// TIA Portal project "Scena_pick_place" (V16)
// Vorlageprojekt für das Buch mit Zielsystem S7-1200

(* hardware
DEVICE "S7-1200-Station_1"  S7-1200 Station
   slot 0: "Baugruppenträger_0"  Rack  V1.0
   slot 1: "PLC_1"  CPU 1211C DC/DC/DC  6ES7 211-1AE40-0XB0  V4.1
*)

// ===== PLC "PLC_1"  CPU 1211C DC/DC/DC =====

VAR_GLOBAL   // PLC tag table "Standard-Variablentabelle"
   "Entry_Conveyor" AT %A0.0 : Bool;
   "Auto" AT %E0.0 : Bool;
   "Emergency_stop" AT %E0.1 : Bool;
   "Item_at_entry" AT %I0.2 : Bool;
   "Item_at_exit" AT %I0.3 : Bool;
   "Item_detected" AT %I0.4 : Bool;
   "Manual" AT %I0.5 : Bool;
   "Moving_x" AT %I0.6 : Bool;
   "Moving_z" AT %I0.7 : Bool;
   "Exit_conveyor" AT %Q0.1 : Bool;
   "Grab" AT %Q0.2 : Bool;
   "Move_x" AT %Q0.3 : Bool;
   "Move_z" AT %Q0.4 : Bool;
   "Reset" AT %I1.0 : Bool;
   "Start" AT %I1.1 : Bool;
   "Stop" AT %I1.2 : Bool;
   "Reset_light" AT %Q0.5 : Bool;
   "Start_light" AT %Q0.6 : Bool;
   "Stop_light" AT %Q0.7 : Bool;
   "Tag_1" AT %M0.0 : Bool;
   "Tag_2" AT %M0.1 : Bool;
   "Tag_3" AT %M0.2 : Bool;
   "Tag_4" AT %M0.3 : Bool;
   "Tag_5" AT %M0.4 : Bool;
   "Tag_6" AT %M0.5 : Bool;
   "Counter" AT %QD30 : DInt;
END_VAR

FUNCTION "MHJ-PLC-Lab-Function-S71200" : Void   // FC9000, SCL
{ S7_Optimized_Access := 'TRUE' }
VERSION : 0.1
   VAR_TEMP
      rdTimeReturn : Int;
      outputTime : DTL;
      SyncVal : Byte;
      forVal : Int;
      forVal_2 : Int;
      Value : Byte;
   END_VAR
   VAR CONSTANT
      CompVal : Byte := 16#34;
      Value_01 : Byte := 16#11;
      Value_01_DW : DWord := 16#A165_D992;
      Value_02_DW : DWord := 16#58BE_4401;
   END_VAR
BEGIN

   #Value:=PEEK(area := 16#82,
        dbNumber := 0,
        byteOffset := 511);
   #Value := #Value + 1;

   POKE(area := 16#82,
        dbNumber := 0,
        byteOffset := 511,
        value := #Value);

   POKE(area:=16#81,
        dbNumber:=0,
        byteOffset:=1016,
        value:=#Value_01_DW);
   POKE(area := 16#81,
        dbNumber := 0,
        byteOffset := 1020,
        value := #Value_02_DW);

   POKE(area := 16#81,
        dbNumber := 0,
        byteOffset := 511,
        value := B#16#00);

   FOR #forVal := 0 TO 120 DO
       FOR #forVal_2:=0 TO 10 DO
           #rdTimeReturn:=RD_SYS_T(#outputTime);
           #rdTimeReturn := WR_SYS_T(#outputTime);
           #rdTimeReturn := RD_SYS_T(#outputTime);
           #rdTimeReturn := WR_SYS_T(#outputTime);
       END_FOR;
       #SyncVal:= PEEK(area := 16#81,
                      dbNumber := 0,
                      byteOffset := 511);
       IF #SyncVal = #CompVal THEN
          GOTO M_1;
       END_IF;
   END_FOR;
   RETURN;

   M_1:
   POKE(area := 16#81,
        dbNumber := 0,
        byteOffset := 511,
        value := B#16#0);
END_FUNCTION

ORGANIZATION_BLOCK "Main"   // OB1, LAD, ProgramCycle
TITLE = "Main Program Sweep (Cycle)"
{ S7_Optimized_Access := 'TRUE' }
VERSION : 0.1
   VAR_INPUT
      Initial_Call : Bool;   // Initial call of this OB
      Remanence : Bool;   // =True, if remanent data are available
   END_VAR
   VAR_TEMP   // added for the SCL form of the ladder/FBD networks
      _w1 : Bool;
   END_VAR
BEGIN

REGION Network 1: Konnektierungsbaustein für PLC-Lab / Connection to Factory
   // Im Netzwerk 1 wird der Konnektierungsbaustein für PLC-Lab aufgerufen.
   // Dieser Aufruf darf nicht entfernt werden!
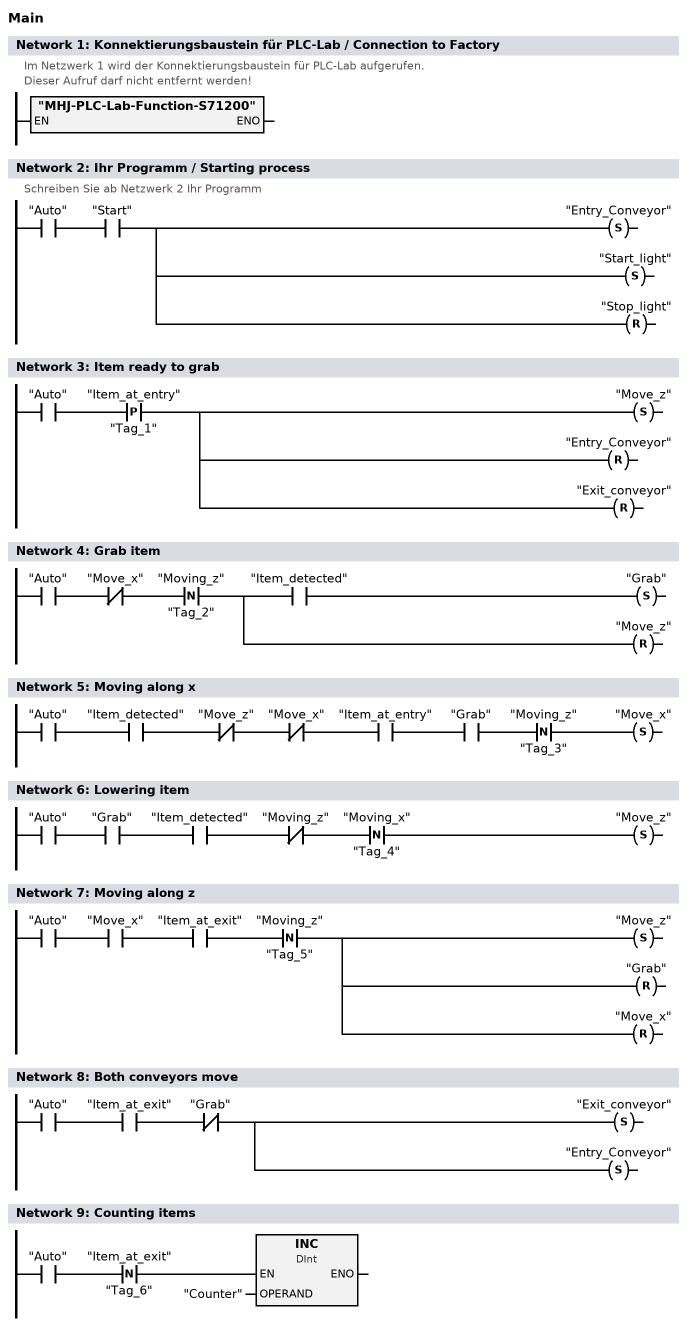
   RUNG wire#powerrail
      "MHJ-PLC-Lab-Function-S71200"()
   END_RUNG
   // the same network as SCL:
   "MHJ-PLC-Lab-Function-S71200"();
END_REGION

REGION Network 2: Ihr Programm / Starting process
   // Schreiben Sie ab Netzwerk 2 Ihr Programm
   RUNG wire#powerrail
      Contact( "Auto" )
      Contact( "Start" )
      wire#w1
      S_Coil( "Entry_Conveyor" )
   END_RUNG
   RUNG wire#w1
      S_Coil( "Start_light" )
   END_RUNG
   RUNG wire#w1
      R_Coil( "Stop_light" )
   END_RUNG
   // the same network as SCL:
   IF "Auto" AND "Start" THEN
       "Entry_Conveyor" := TRUE;
       "Start_light" := TRUE;
       "Stop_light" := FALSE;
   END_IF;
END_REGION

REGION Network 3: Item ready to grab
   RUNG wire#powerrail
      Contact( "Auto" )
      P_Contact(operand := "Item_at_entry", bit := "Tag_1")
      wire#w1
      S_Coil( "Move_z" )
   END_RUNG
   RUNG wire#w1
      R_Coil( "Entry_Conveyor" )
   END_RUNG
   RUNG wire#w1
      R_Coil( "Exit_conveyor" )
   END_RUNG
   // the same network as SCL:
   #_w1 := "Auto" AND "Item_at_entry" AND NOT "Tag_1";   // rising edge of "Item_at_entry"
   "Tag_1" := "Item_at_entry";
   IF #_w1 THEN
       "Move_z" := TRUE;
       "Entry_Conveyor" := FALSE;
       "Exit_conveyor" := FALSE;
   END_IF;
END_REGION

REGION Network 4: Grab item
   RUNG wire#powerrail
      Contact( "Auto" )
      I_Contact( "Move_x" )
      N_Contact(operand := "Moving_z", bit := "Tag_2")
      wire#w1
      Contact( "Item_detected" )
      S_Coil( "Grab" )
   END_RUNG
   RUNG wire#w1
      R_Coil( "Move_z" )
   END_RUNG
   // the same network as SCL:
   #_w1 := "Auto" AND NOT "Move_x" AND NOT "Moving_z" AND "Tag_2";   // falling edge of "Moving_z"
   "Tag_2" := "Moving_z";
   IF #_w1 AND "Item_detected" THEN "Grab" := TRUE; END_IF;
   IF #_w1 THEN "Move_z" := FALSE; END_IF;
END_REGION

REGION Network 5: Moving along x
   RUNG wire#powerrail
      Contact( "Auto" )
      Contact( "Item_detected" )
      I_Contact( "Move_z" )
      I_Contact( "Move_x" )
      Contact( "Item_at_entry" )
      Contact( "Grab" )
      N_Contact(operand := "Moving_z", bit := "Tag_3")
      S_Coil( "Move_x" )
   END_RUNG
   // the same network as SCL:
   #_w1 := "Auto" AND "Item_detected" AND NOT "Move_z" AND NOT "Move_x" AND "Item_at_entry" AND "Grab" AND NOT "Moving_z" AND "Tag_3";   // falling edge of "Moving_z"
   "Tag_3" := "Moving_z";
   IF #_w1 THEN "Move_x" := TRUE; END_IF;
END_REGION

REGION Network 6: Lowering item
   RUNG wire#powerrail
      Contact( "Auto" )
      Contact( "Grab" )
      Contact( "Item_detected" )
      I_Contact( "Moving_z" )
      N_Contact(operand := "Moving_x", bit := "Tag_4")
      S_Coil( "Move_z" )
   END_RUNG
   // the same network as SCL:
   #_w1 := "Auto" AND "Grab" AND "Item_detected" AND NOT "Moving_z" AND NOT "Moving_x" AND "Tag_4";   // falling edge of "Moving_x"
   "Tag_4" := "Moving_x";
   IF #_w1 THEN "Move_z" := TRUE; END_IF;
END_REGION

REGION Network 7: Moving along z
   RUNG wire#powerrail
      Contact( "Auto" )
      Contact( "Move_x" )
      Contact( "Item_at_exit" )
      N_Contact(operand := "Moving_z", bit := "Tag_5")
      wire#w1
      S_Coil( "Move_z" )
   END_RUNG
   RUNG wire#w1
      R_Coil( "Grab" )
   END_RUNG
   RUNG wire#w1
      R_Coil( "Move_x" )
   END_RUNG
   // the same network as SCL:
   #_w1 := "Auto" AND "Move_x" AND "Item_at_exit" AND NOT "Moving_z" AND "Tag_5";   // falling edge of "Moving_z"
   "Tag_5" := "Moving_z";
   IF #_w1 THEN
       "Move_z" := TRUE;
       "Grab" := FALSE;
       "Move_x" := FALSE;
   END_IF;
END_REGION

REGION Network 8: Both conveyors move
   RUNG wire#powerrail
      Contact( "Auto" )
      Contact( "Item_at_exit" )
      I_Contact( "Grab" )
      wire#w1
      S_Coil( "Exit_conveyor" )
   END_RUNG
   RUNG wire#w1
      S_Coil( "Entry_Conveyor" )
   END_RUNG
   // the same network as SCL:
   IF "Auto" AND "Item_at_exit" AND NOT "Grab" THEN
       "Exit_conveyor" := TRUE;
       "Entry_Conveyor" := TRUE;
   END_IF;
END_REGION

REGION Network 9: Counting items
   RUNG wire#powerrail
      Contact( "Auto" )
      N_Contact(operand := "Item_at_exit", bit := "Tag_6")
      { S7_Templates := "DestType := DInt" } Inc( "Counter" )
   END_RUNG
   // the same network as SCL:
   #_w1 := "Auto" AND NOT "Item_at_exit" AND "Tag_6";   // falling edge of "Item_at_exit"
   "Tag_6" := "Item_at_exit";
   IF #_w1 THEN "Counter" := "Counter" + 1; END_IF;
END_REGION
END_ORGANIZATION_BLOCK